// TIA Portal V19 export
FUNCTION "LAF_ManualOperationLine_Notes" : Void   // FC23, LAD
TITLE = LAF_ManualOperationLine_Notes
// Here are some points that are important for the use and configuration of manual operation lines:
// 
// * For the appearance of each Line, Json files with the configurations need to be added manually to the target machine. Be it in a PC Runtime or Panel. The Path is set in the HMI as the HMI Tag "manualOperationFilePath" in the "03_manualOperation" table. We have set it to "D:\\JsonFiles\\". The files used for this example are saved in the project UserFiles. The Path for the Panel can look like "/home/industrial/JsonFiles".
// 
// * Under "CallManualOperationLines" are the calls for the main configuration of a Equipment module and the control of each line.
//  * Each Equipment module needs to have a defined number. For the numeration we recommend using the second and third digit for the Equipment module number used in the project and the fourth digit with the number of the unit.
// 
// * The texts for the Areas are defined as text lists in the HMI. For the corresponding group, the naming is currently set as "EquipmentAreas_XXXX" with the XXXX as the Equipment Module number. It is set in the "manualOperationEm.equipmentModuleNum".
//  
// * There can be defined 16 color text lists. Each text list defines: "1 - normal, 2 - pressed, 3 - confirmed, 4 - deactivated, 5 - deactivated+pressed".
//  * The color value is in hex with the 2 first values on the left defining the transparency and the rest as normal color values.
//  * The text list name is currently "LAF_manualColorX" with the X as the text list number.
// 
// * If another HMI device is added, please don't forget the Scheduled tasks for updating the lines  
// 
// * The amount of areas is defined by the size of the array in the configuration of areas. The array should start.
// stored: SetENOAutomatically false
BEGIN
END_FUNCTION
